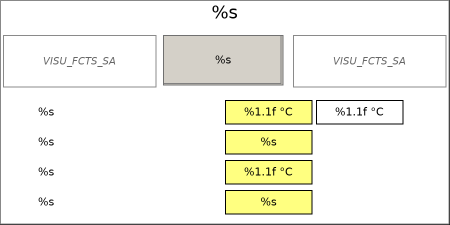
VISUALIZATION SA_HEATING  // 450x225
VAR_IN_OUT
	m_Input_UserRight:	BOOL;
	m_Input_Machine:	BLOCK_MODE_MARCHE_V2_0;
	m_Input_PRG:		BLOCK_PRG_CHAUFFAGE;
END_VAR
    Rectangle (0,0 450x225), "%s", text list: 'TextList_Navigation', text index: 10
    Frame (3,35 153x52)
        shows VISU_FCTS_SA(m_Input_ID_XML := 24, m_Input_UserRight := PRG_USER.ACTU_USER.FONCTION_SA, m_Input_Operation := m_Input_PRG.CHAUFFAGE.OP_MARCHE)
    Frame (293,35 153x52)
        shows VISU_FCTS_SA(m_Input_ID_XML := 25, m_Input_UserRight := PRG_USER.ACTU_USER.FONCTION_SA, m_Input_Operation := m_Input_PRG.CHAUFFAGE.OP_ARRET)
    Button (163,35 120x50), "%s", input disabled if: (NOT PRG_USER.ACTU_USER.FONCTION_SA AND NOT m_Input_Machine.STATE_Prod) OR (NOT PRG_USER.ACTU_USER.MODIF_ENLIGNE AND m_Input_Machine.STATE_Prod), text list: 'TextList_Basiques', text index: 19
        tap m_Input_PRG.CHAUFFAGE.CO_Modif
    Rectangle (35,100 188x24), "%s", text list: 'TextList_Chauffage', text index: 9
    RoundedRectangle (316,100 87x24), "%1.1f °C", text variable: m_Input_PRG.CHAUFFAGE.CH.IN_Temperature
    RoundedRectangle (225,100 87x24), "%1.1f °C", text variable: m_Input_PRG.CHAUFFAGE.PRM_Temp, input disabled if: (NOT PRG_USER.ACTU_USER.FONCTION_SA AND NOT m_Input_Machine.STATE_Prod) OR (NOT PRG_USER.ACTU_USER.MODIF_ENLIGNE AND m_Input_Machine.STATE_Prod)
        OnMouseClick: write the text variable via VisuDialogs.Numpad, min 20, max m_Input_PRG.PRM_Max_Temp
    Rectangle (35,130 188x24), "%s", text list: 'TextList_Chauffage', text index: 6
    RoundedRectangle (225,130 87x24), "%s", text variable: m_Input_PRG.CHAUFFAGE.PRM_Tps_Stab, input disabled if: (NOT PRG_USER.ACTU_USER.FONCTION_SA AND NOT m_Input_Machine.STATE_Prod) OR (NOT PRG_USER.ACTU_USER.MODIF_ENLIGNE AND m_Input_Machine.STATE_Prod)
        OnMouseClick: write the text variable via VisuDialogs.Keypad
    Rectangle (35,160 188x24), "%s", text list: 'TextList_Chauffage', text index: 10
    RoundedRectangle (225,160 87x24), "%1.1f °C", text variable: m_Input_PRG.CHAUFFAGE.PRM_Delta_Stab, input disabled if: (NOT PRG_USER.ACTU_USER.FONCTION_SA AND NOT m_Input_Machine.STATE_Prod) OR (NOT PRG_USER.ACTU_USER.MODIF_ENLIGNE AND m_Input_Machine.STATE_Prod)
        OnMouseClick: write the text variable via VisuDialogs.Numpad, min 0, max 50
    Rectangle (35,190 188x24), "%s", text list: 'TextList_Chauffage', text index: 8
    RoundedRectangle (225,190 87x24), "%s", text variable: m_Input_PRG.CHAUFFAGE.DEF_Stab.DELAY, input disabled if: (NOT PRG_USER.ACTU_USER.FONCTION_SA AND NOT m_Input_Machine.STATE_Prod) OR (NOT PRG_USER.ACTU_USER.MODIF_ENLIGNE AND m_Input_Machine.STATE_Prod)
        OnMouseClick: write the text variable via VisuDialogs.Keypad
END_VISUALIZATION

(* stored: Version 1.1.0.1, ProductVersion 3.1.4024.10
   Visu SA_HEATING: Id {981ee1cc-d798-41ee-a3bc-7ce9209e26a0} *)
